// TIA Portal V20 export
DATA_BLOCK "instFB_AxisCtrl"   // DB2
VERSION : 1.1
// stored: InstanceOfName FB_AxisCtrl, InstanceOfType FB
"FB_AxisCtrl"
   // VAR
   //    instPower_J1 { S7_SetPoint := 'True'} : MC_POWER;
   //    instPower_J2 { S7_SetPoint := 'True'} : MC_POWER;
   //    instPower_J3 { S7_SetPoint := 'True'} : MC_POWER;
   //    instPower_J4 { S7_SetPoint := 'True'} : MC_POWER;
   //    instHome_J1 { S7_SetPoint := 'True'} : MC_HOME;
   //    instHome_J2 { S7_SetPoint := 'True'} : MC_HOME;
   //    instHome_J3 { S7_SetPoint := 'True'} : MC_HOME;
   //    instHome_J4 { S7_SetPoint := 'True'} : MC_HOME;
   //    instReset_J1 { S7_SetPoint := 'True'} : MC_RESET;
   //    instReset_J2 { S7_SetPoint := 'True'} : MC_RESET;
   //    instReset_J3 { S7_SetPoint := 'True'} : MC_RESET;
   //    instReset_J4 { S7_SetPoint := 'True'} : MC_RESET;
   //    instReset_Kin { S7_SetPoint := 'True'} : MC_RESET;
   // END_VAR
BEGIN
END_DATA_BLOCK
